PROGRAM GarageDoor
VAR
	bActuationButton AT %I* : BOOL; //actuation button connected through visualization
	bOpenSensor AT %Q* : BOOL;
	bClosedSensor AT %Q* : BOOL; //sensor conected to lights 
	bDriveOverloadSensor : BOOL; //sensor that indicates if there is an error
	bLightForMotion : BOOL; // light that turns on if the door is in motion
	fbGarage : OpenCloseGarage;
	bVisualizationOpenClose : BOOL;
	bPauseLight AT %Q* : BOOL; //light that blinks if the door is paused
	bErrorButton AT %I* : BOOL; //button that puts the door in error
END_VAR

fbGarage.bActuationProgram := bActuationButton; //we activate the garage

bOpenSensor := fbGarage.bDoorOpen;
bClosedSensor := fbGarage.bDoorClosed;
bDriveOverloadSensor := fbGarage.bDriveOverload; //we set the sensors

bLightForMotion := fbGarage.bLight;
bVisualizationOpenClose := fbGarage.bVisualization;


bPauseLight := fbGarage.bLightForPause;

fbGarage.bError := bErrorButton;



fbGarage();

END_PROGRAM

(* stored: Version 1.1.0.1, ProductVersion 3.1.4024.12
   POU GarageDoor: Id {73ceeb09-c68d-4e8a-b7f3-60ed11bd254d}, SpecialFunc None *)
